PROGRAM P_BACnet_Level
VAR
	ton_DelayForBACnet		: TON;
END_VAR

//keep BACnet object alive
fbBACnet_AV_SL_Level_1(Device := Device, bEnablePV := TRUE, bNullPV := FALSE);
fbBACnet_AV_SL_Level_2(Device := Device, bEnablePV := TRUE, bNullPV := FALSE);
fbBACnet_AV_SL_Level_3(Device := Device, bEnablePV := TRUE, bNullPV := FALSE);
fbBACnet_AV_SL_Level_4(Device := Device, bEnablePV := TRUE, bNullPV := FALSE);
fbBACnet_AV_SL_Level_5(Device := Device, bEnablePV := TRUE, bNullPV := FALSE);
fbBACnet_AV_SL_Level_6(Device := Device, bEnablePV := TRUE, bNullPV := FALSE);
fbBACnet_AV_SL_Level_7(Device := Device, bEnablePV := TRUE, bNullPV := FALSE);
fbBACnet_AV_SL_Level_8(Device := Device, bEnablePV := TRUE, bNullPV := FALSE);
fbBACnet_AV_SL_Level_9(Device := Device, bEnablePV := TRUE, bNullPV := FALSE);
fbBACnet_AV_SL_Level_10(Device := Device, bEnablePV := TRUE, bNullPV := FALSE);

//if Reset was not called
IF NOT bBACnet_ResetManual AND NOT bBACnet_SetManual THEN
	//if lamp is in manual mode, assign BACnet fPresentValue to nLevel
	IF GVL_IO.arrStreetLamps[1].bManualCtrl  THEN GVL_IO.arrStreetLamps[1].nLevel  := REAL_TO_BYTE(fbBACnet_AV_SL_Level_1.fPresentValue);  END_IF
	IF GVL_IO.arrStreetLamps[2].bManualCtrl  THEN GVL_IO.arrStreetLamps[2].nLevel  := REAL_TO_BYTE(fbBACnet_AV_SL_Level_2.fPresentValue);  END_IF
	IF GVL_IO.arrStreetLamps[3].bManualCtrl  THEN GVL_IO.arrStreetLamps[3].nLevel  := REAL_TO_BYTE(fbBACnet_AV_SL_Level_3.fPresentValue);  END_IF
	IF GVL_IO.arrStreetLamps[4].bManualCtrl  THEN GVL_IO.arrStreetLamps[4].nLevel  := REAL_TO_BYTE(fbBACnet_AV_SL_Level_4.fPresentValue);  END_IF
	IF GVL_IO.arrStreetLamps[5].bManualCtrl  THEN GVL_IO.arrStreetLamps[5].nLevel  := REAL_TO_BYTE(fbBACnet_AV_SL_Level_5.fPresentValue);  END_IF
	IF GVL_IO.arrStreetLamps[6].bManualCtrl  THEN GVL_IO.arrStreetLamps[6].nLevel  := REAL_TO_BYTE(fbBACnet_AV_SL_Level_6.fPresentValue);  END_IF
	IF GVL_IO.arrStreetLamps[7].bManualCtrl  THEN GVL_IO.arrStreetLamps[7].nLevel  := REAL_TO_BYTE(fbBACnet_AV_SL_Level_7.fPresentValue);  END_IF
	IF GVL_IO.arrStreetLamps[8].bManualCtrl  THEN GVL_IO.arrStreetLamps[8].nLevel  := REAL_TO_BYTE(fbBACnet_AV_SL_Level_8.fPresentValue);  END_IF
	IF GVL_IO.arrStreetLamps[9].bManualCtrl  THEN GVL_IO.arrStreetLamps[9].nLevel  := REAL_TO_BYTE(fbBACnet_AV_SL_Level_9.fPresentValue);  END_IF
	IF GVL_IO.arrStreetLamps[10].bManualCtrl THEN GVL_IO.arrStreetLamps[10].nLevel := REAL_TO_BYTE(fbBACnet_AV_SL_Level_10.fPresentValue); END_IF
END_IF

END_PROGRAM

(* stored: Version 1.1.0.1, ProductVersion 3.1.4024.5
   POU P_BACnet_Level: Id {adbf72dc-6ab6-4f9e-a501-48ed86d435f9}, SpecialFunc None *)
